// TIA Portal V21 export
FUNCTION_BLOCK "FB311"   // FB311, LAD
TITLE = FB311
{ S7_Optimized_Access := 'TRUE' }
AUTHOR : PRECISE
FAMILY : PRECISE
// TEMPERATURE CONTROL
// stored: AutoNumber false, MemoryReserve 100, SetENOAutomatically false
   VAR_INPUT
      Enable : Bool;
      Disable : Bool;
      Fault : Bool;
      SecPulse : Bool;
      AlwaysTrue : Bool;
      StartConfirmationPopupSel : Bool;   // StartConfirmationPopupSel: 0-NO/1-YES
      EndConfirmationPopupSel : Bool;   // EndConfirmationPopupSel: 0-NO/1-YES
      TimebaseSel : Bool;   // Timebase Selection: 0-sec/1-min
      TemperatureMaintainSel : Bool;   // Temperature Maintain Selection: 0-NO/1-YES
      BypassSel : Bool;   // Bypass Selection: 0-NO/1-YES
      JacketAirPurgingSel : Bool;   // Applicable for if Air Inlet Valve is present in jacket. 0-NO/1-YES
      TemperatureControlSel : Int;   // Temperature Control Sel : 0-Heat/1-Cool
      SensorSel : Int;   // Sensor Slection: 0-Vessel/1-Jacket
      BatchSizeSel : Int;   // Batch Size Sel:0-Small/1-Big
      HeatingUtilitySel : Int;   // Heating Utility Selection: 0-Steam/1-Hot Water
      CoolingUtilitySelection : Int;   // 0-cooling/1-chilling/2-brine/3-cooling+chilling/4-chilling+brine/5-cooling+chilling+Brine
      SetTemperature : Real := 60.0;
      TimeMin : Int := 1;   // For Temperature Maintain Selection: 1-YES & Bypass Selection: 1-YES
      TimeSec : Int := 30;   // For Temperature Maintain Selection: 1-YES & Bypass Selection: 0-NO
      ActualTemperatureVessel : Real;   // For Sensor Slection: 0-Vessel
      ActualTemperatureJacket : Real;   // For Sensor Slection: 1-Jacket
      JVDelay : Int := 5;
      JDDelay : Int := 5;
      TemperatureTol : Real := 0.3;
      CoolingThreshold : Real := 25.0;   // Temperature to change utility from cooling water to chilled water
      ChillingThreshold : Real := 15.0;   // Temperature to change utility from chilled water to brine water
      HeatHighTemperatureTol : Real := 3.0;
      CoolLowTemperatureTol : Real := 3.0;
      JacketAirPurgingTimeSec : Int := 10;
   END_VAR
   VAR_OUTPUT
      JacketAirValve : Bool;
      BypassValve : Bool;
      JacketVentValve1 : Bool;
      JacketDrainValve1 : Bool;
      CoolingWaterInletValve1 : Bool;
      CoolingWaterOutletValve1 : Bool;
      ChilledWaterInletValve1 : Bool;
      ChilledWaterOutletValve1 : Bool;
      BrineWaterInletValve1 : Bool;
      BrineWaterOutletValve1 : Bool;
      HotWaterInletValve1 : Bool;
      HotWaterOutletValve1 : Bool;
      SteamInlet1 : Bool;
      Condensateoutlet1 : Bool;
      JacketVentValve2 : Bool;
      JacketDrainValve2 : Bool;
      CoolingWaterInletValve2 : Bool;
      CoolingWaterOutletValve2 : Bool;
      ChilledWaterInletValve2 : Bool;
      ChilledWaterOutletValve2 : Bool;
      BrineWaterInletValve2 : Bool;
      BrineWaterOutletValve2 : Bool;
      HotWaterInletValve2 : Bool;
      HotWaterOutletValve2 : Bool;
      SteamInlet2 : Bool;
      Condensateoutlet2 : Bool;
      AlarmHeatHighTemperature : Bool;
      AlarmCoolLowTemperature : Bool;
      StartConfirmationPopup : Bool;   // For Start Confirmation Popup Selection: Yes
      EndConfirmationPopup : Bool;   // For End Confirmation Popup Selection: Yes
      JacketAirPurgingPopup : Bool;
      TimeMinPV : DInt;
      TimeSecPV : DInt;
      JacketAirPurgingTimeSecPV : Int;
      PrintTrigger : Bool;
      PrintWord : Int;
      PrintStatus : String[50];
   END_VAR
   VAR_IN_OUT
      Start : Bool;
      Stop : Bool;
      Reset : Bool;
      StartConfirmationAck : Bool;   // For Start Confirmation Popup Selection: Yes
      EndConfirmationAck : Bool;   // For End Confirmation Popup Selection: Yes
      JacketAirPurgingAck : Bool;
      AlarmAck : Bool;
      SpareBtn1 : Bool;
      Running : Bool;
      Selected : Bool;
      Paused : Bool;
      StartConfirmationPopupTemp : Bool;   // For Start Confirmation Popup Selection: Yes
      EndConfirmationPopupTemp : Bool;   // For End Confirmation Popup Selection: Yes
      Started : Bool;
      Over : Bool;
      StartJVDelay : Bool;
      StartJDDelay : Bool;
      StartUtility : Bool;
      StartChilling : Bool;
      StartBrine : Bool;
      StartJacketAirPurging : Bool;
      HeatTempReached : Bool;
      CoolTempReached : Bool;
      TemperatureTolNeg : Real;
      TemperatureTolPos : Real;
      HeatHighTemperatureTolCal : Real := 3.0;
      CoolLowTemperatureTolCal : Real := 3.0;
      JacketPressureSelection : Bool;   // 0-no,1-yes
      JacketPressureReached : Bool;
      JacketUtilityPressureValve : Bool;
      JAcketAlarms : Bool;
      Temp : Bool;
      JacketTime : Int;
      JacketSafetyPressure : Real;
      JAcketActPressure : Real;
   END_VAR
   VAR
      PrintTriggerTemp : Bool;
      RE1 : Bool;
      RE2 : Bool;
      RE3 : Bool;
      RE4 : Bool;
      RE5 : Bool;
      RE6 : Bool;
      RE7 : Bool;
      RE8 : Bool;
      RE9 : Bool;
      RE10 : Bool;
      RE11 : Bool;
      "Timer" : "FB101";
      PrintTriggerResetTimer { S7_SetPoint := 'True'} : TON_TIME;
      BtnResetTimer { S7_SetPoint := 'True'} : TON_TIME;
      JVDelayTime { S7_SetPoint := 'True'} : "FB103";
      JDDelayTime { S7_SetPoint := 'True'} : "FB103";
      JAPTime { S7_SetPoint := 'True'} : "FB103";
      ActualTemperature : Real;
      JacketpressureTimer { S7_SetPoint := 'True'} : "FB103";
      FB101_Instance { S7_SetPoint := 'True'} : "FB101";
   END_VAR
   VAR_TEMP
      STATUS1 : String[40];
      STATUS2 : String[40];
      STATUS3 : String[40];
      STATUS4 : String[40];
      STATUS5 : String[40];
      STATUS6 : String[40];
   END_VAR
   VAR_TEMP   // added for the SCL form of the ladder/FBD networks
      _w1 : Bool;
      _w2 : Bool;
      _w3 : Bool;
      _w4 : Bool;
      _w5 : Bool;
      _w6 : Bool;
      _w7 : Bool;
      _w8 : Bool;
   END_VAR
BEGIN

REGION Network 1: Running
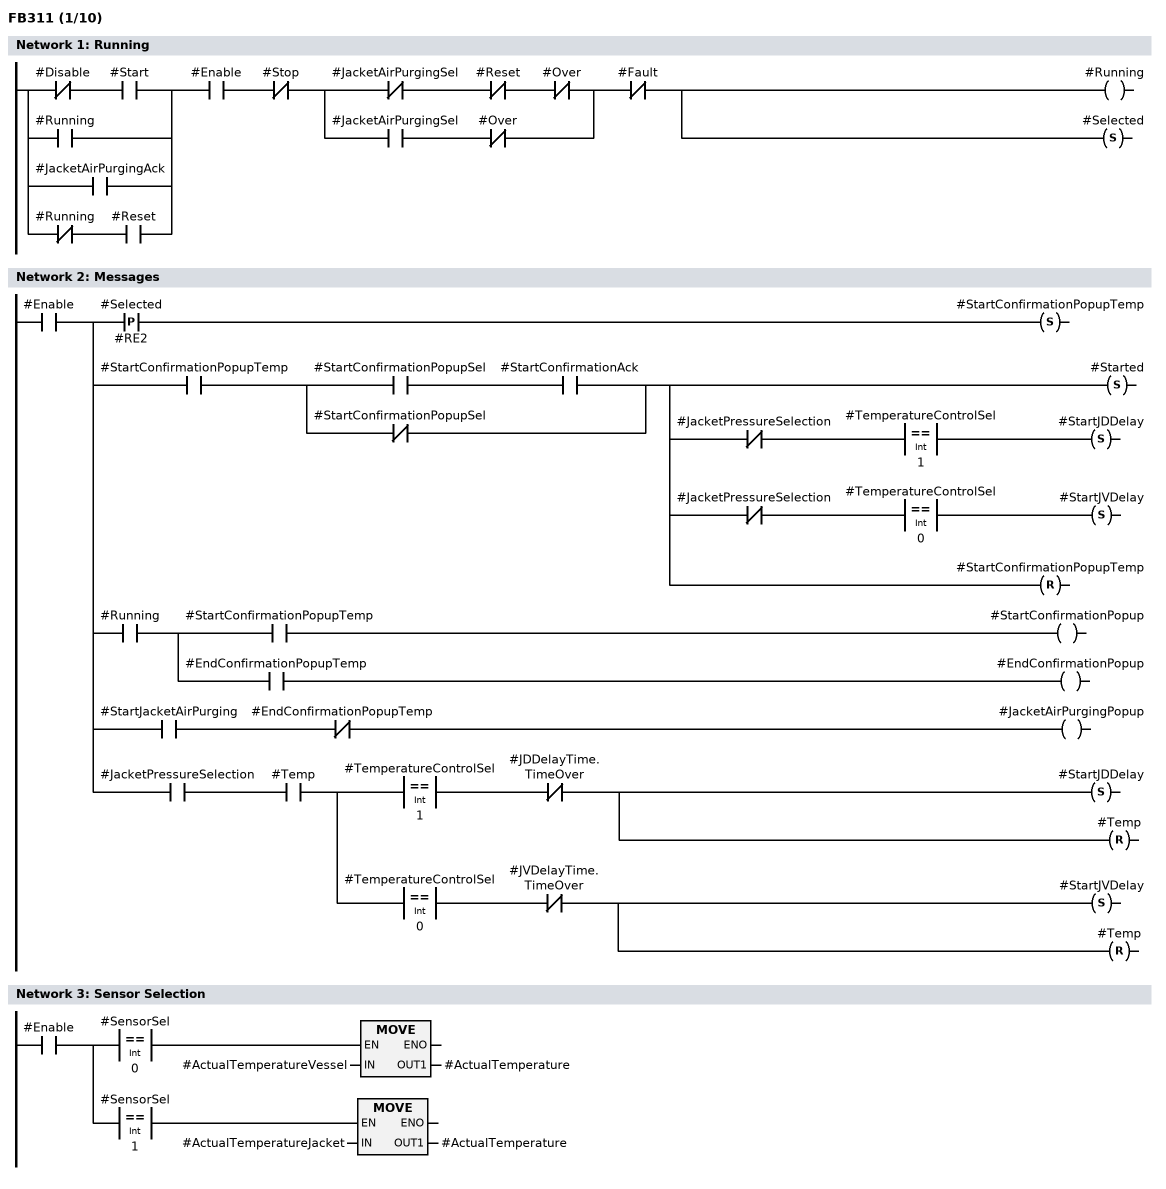
   RUNG wire#powerrail
      I_Contact( #Disable )
      Contact( #Start )
      wire#w1
      Contact( #Enable )
      I_Contact( #Stop )
      wire#w2
      I_Contact( #JacketAirPurgingSel )
      I_Contact( #Reset )
      I_Contact( #Over )
      wire#w3
      I_Contact( #Fault )
      wire#w4
      Coil( #Running )
   END_RUNG
   RUNG wire#powerrail
      Contact( #Running )
   END_RUNG wire#w1
   RUNG wire#powerrail
      Contact( #JacketAirPurgingAck )
   END_RUNG wire#w1
   RUNG wire#powerrail
      I_Contact( #Running )
      Contact( #Reset )
   END_RUNG wire#w1
   RUNG wire#w2
      Contact( #JacketAirPurgingSel )
      I_Contact( #Over )
   END_RUNG wire#w3
   RUNG wire#w4
      S_Coil( #Selected )
   END_RUNG
   // the same network as SCL:
   #Running := ((NOT #Disable AND #Start) OR #Running OR #JacketAirPurgingAck OR (NOT #Running AND #Reset)) AND #Enable AND NOT #Stop AND ((NOT #JacketAirPurgingSel AND NOT #Reset AND NOT #Over) OR (#JacketAirPurgingSel AND NOT #Over)) AND NOT #Fault;
   IF #Running THEN #Selected := TRUE; END_IF;
END_REGION

REGION Network 2: Messages
   RUNG wire#powerrail
      Contact( #Enable )
      wire#w1
      P_Contact(operand := #Selected, bit := #RE2)
      S_Coil( #StartConfirmationPopupTemp )
   END_RUNG
   RUNG wire#w1
      Contact( #StartConfirmationPopupTemp )
      wire#w2
      Contact( #StartConfirmationPopupSel )
      Contact( #StartConfirmationAck )
      wire#w3
      S_Coil( #Started )
   END_RUNG
   RUNG wire#w2
      I_Contact( #StartConfirmationPopupSel )
   END_RUNG wire#w3
   RUNG wire#w3
      I_Contact( #JacketPressureSelection )
      { S7_Templates := "SrcType := Int" } EQ_Contact(in1 := #TemperatureControlSel, in2 := 1)
      S_Coil( #StartJDDelay )
   END_RUNG
   RUNG wire#w3
      I_Contact( #JacketPressureSelection )
      { S7_Templates := "SrcType := Int" } EQ_Contact(in1 := #TemperatureControlSel, in2 := 0)
      S_Coil( #StartJVDelay )
   END_RUNG
   RUNG wire#w3
      R_Coil( #StartConfirmationPopupTemp )
   END_RUNG
   RUNG wire#w1
      Contact( #Running )
      wire#w4
      Contact( #StartConfirmationPopupTemp )
      Coil( #StartConfirmationPopup )
   END_RUNG
   RUNG wire#w4
      Contact( #EndConfirmationPopupTemp )
      Coil( #EndConfirmationPopup )
   END_RUNG
   RUNG wire#w1
      Contact( #StartJacketAirPurging )
      I_Contact( #EndConfirmationPopupTemp )
      Coil( #JacketAirPurgingPopup )
   END_RUNG
   RUNG wire#w1
      Contact( #JacketPressureSelection )
      Contact( #Temp )
      wire#w5
      { S7_Templates := "SrcType := Int" } EQ_Contact(in1 := #TemperatureControlSel, in2 := 1)
      I_Contact( #JDDelayTime.TimeOver )
      wire#w6
      S_Coil( #StartJDDelay )
   END_RUNG
   RUNG wire#w6
      R_Coil( #Temp )
   END_RUNG
   RUNG wire#w5
      { S7_Templates := "SrcType := Int" } EQ_Contact(in1 := #TemperatureControlSel, in2 := 0)
      I_Contact( #JVDelayTime.TimeOver )
      wire#w7
      S_Coil( #StartJVDelay )
   END_RUNG
   RUNG wire#w7
      R_Coil( #Temp )
   END_RUNG
   // the same network as SCL:
   #_w1 := #Enable AND #Selected AND NOT #RE2;   // rising edge of #Selected
   #RE2 := #Selected;
   IF #_w1 THEN #StartConfirmationPopupTemp := TRUE; END_IF;
   #_w2 := #Enable AND #StartConfirmationPopupTemp AND ((#StartConfirmationPopupSel AND #StartConfirmationAck) OR NOT #StartConfirmationPopupSel);
   IF #_w2 THEN #Started := TRUE; END_IF;
   IF #_w2 AND NOT #JacketPressureSelection AND (#TemperatureControlSel = 1) THEN
       #StartJDDelay := TRUE;
   END_IF;
   IF #_w2 AND NOT #JacketPressureSelection AND (#TemperatureControlSel = 0) THEN
       #StartJVDelay := TRUE;
   END_IF;
   IF #_w2 THEN #StartConfirmationPopupTemp := FALSE; END_IF;
   #_w3 := #Enable AND #Running;
   #StartConfirmationPopup := #_w3 AND #StartConfirmationPopupTemp;
   #EndConfirmationPopup := #_w3 AND #EndConfirmationPopupTemp;
   #JacketAirPurgingPopup := #Enable AND #StartJacketAirPurging AND NOT #EndConfirmationPopupTemp;
   #_w4 := #Enable AND #JacketPressureSelection AND #Temp;
   IF #_w4 AND (#TemperatureControlSel = 1) AND NOT #JDDelayTime.TimeOver THEN
       #StartJDDelay := TRUE;
       #Temp := FALSE;
   END_IF;
   IF #_w4 AND (#TemperatureControlSel = 0) AND NOT #JVDelayTime.TimeOver THEN
       #StartJVDelay := TRUE;
       #Temp := FALSE;
   END_IF;
END_REGION

REGION Network 3: Sensor Selection
   RUNG wire#powerrail
      Contact( #Enable )
      wire#w1
      { S7_Templates := "SrcType := Int" } EQ_Contact(in1 := #SensorSel, in2 := 0)
      Move(in := #ActualTemperatureVessel, out1 => #ActualTemperature)
   END_RUNG
   RUNG wire#w1
      { S7_Templates := "SrcType := Int" } EQ_Contact(in1 := #SensorSel, in2 := 1)
      Move(in := #ActualTemperatureJacket, out1 => #ActualTemperature)
   END_RUNG
   // the same network as SCL:
   IF #Enable AND (#SensorSel = 0) THEN #ActualTemperature := #ActualTemperatureVessel; END_IF;
   IF #Enable AND (#SensorSel = 1) THEN #ActualTemperature := #ActualTemperatureJacket; END_IF;
END_REGION

REGION Network 4: Tolerance
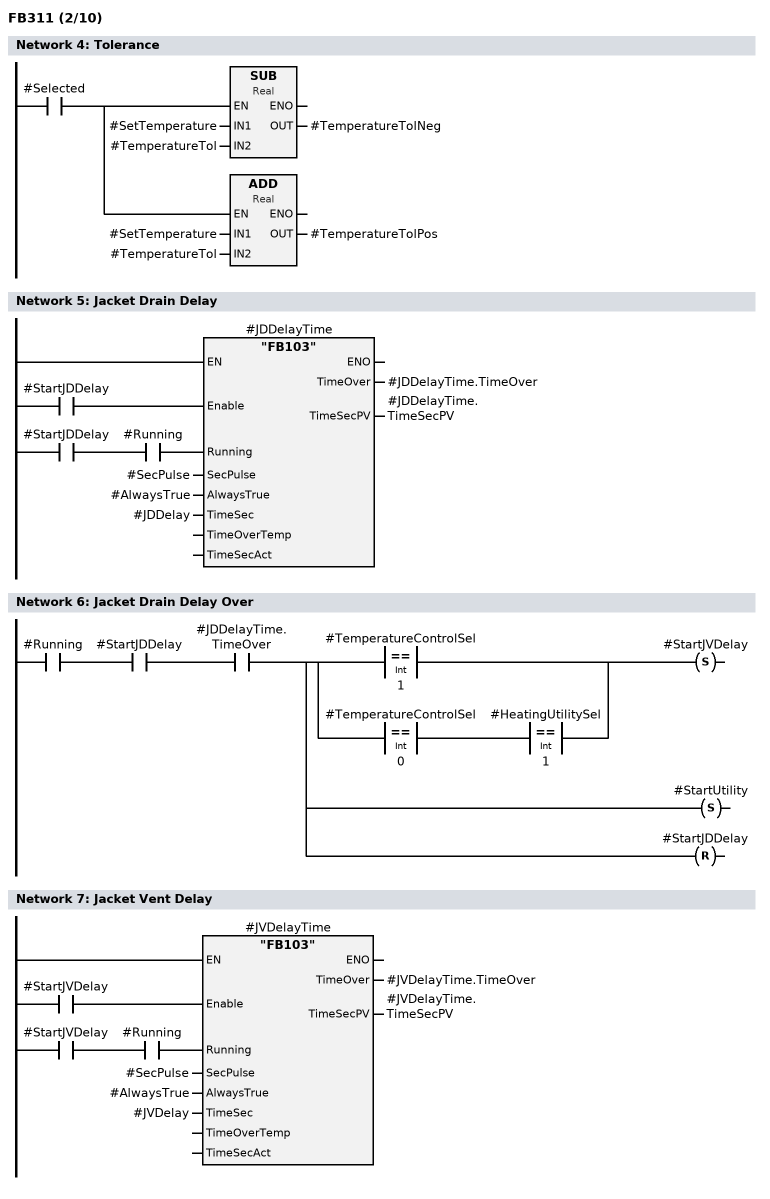
   RUNG wire#powerrail
      Contact( #Selected )
      wire#w1
      { S7_Templates := "SrcType := Real"; S7_GenerateENO := "TRUE" } Sub(in1 := #SetTemperature, in2 := #TemperatureTol, out => #TemperatureTolNeg)
   END_RUNG
   RUNG wire#w1
      { S7_Templates := "SrcType := Real"; S7_GenerateENO := "TRUE" } Add(in1 := #SetTemperature, in2 := #TemperatureTol, out => #TemperatureTolPos)
   END_RUNG
   // the same network as SCL:
   IF #Selected THEN
       #TemperatureTolNeg := #SetTemperature - #TemperatureTol;
       #TemperatureTolPos := #SetTemperature + #TemperatureTol;
   END_IF;
END_REGION

REGION Network 5: Jacket Drain Delay
   RUNG wire#powerrail
      #JDDelayTime(Enable := wire#w1, Running := wire#w2, SecPulse := #SecPulse, AlwaysTrue := #AlwaysTrue, TimeSec := #JDDelay, TimeOverTemp :=, TimeSecAct :=, TimeOver => #JDDelayTime.TimeOver, TimeSecPV => #JDDelayTime.TimeSecPV)
   END_RUNG
   RUNG wire#powerrail
      Contact( #StartJDDelay )
   END_RUNG wire#w1
   RUNG wire#powerrail
      Contact( #StartJDDelay )
      Contact( #Running )
   END_RUNG wire#w2
   // the same network as SCL:
   #JDDelayTime(Enable := #StartJDDelay,   // "FB103"
                Running := #StartJDDelay AND #Running,
                SecPulse := #SecPulse,
                AlwaysTrue := #AlwaysTrue,
                TimeSec := #JDDelay,
                TimeOver => #JDDelayTime.TimeOver,
                TimeSecPV => #JDDelayTime.TimeSecPV);
END_REGION

REGION Network 6: Jacket Drain Delay Over
   RUNG wire#powerrail
      Contact( #Running )
      Contact( #StartJDDelay )
      Contact( #JDDelayTime.TimeOver )
      wire#w1
      { S7_Templates := "SrcType := Int" } EQ_Contact(in1 := #TemperatureControlSel, in2 := 1)
      wire#w2
      S_Coil( #StartJVDelay )
   END_RUNG
   RUNG wire#w1
      { S7_Templates := "SrcType := Int" } EQ_Contact(in1 := #TemperatureControlSel, in2 := 0)
      { S7_Templates := "SrcType := Int" } EQ_Contact(in1 := #HeatingUtilitySel, in2 := 1)
   END_RUNG wire#w2
   RUNG wire#w1
      S_Coil( #StartUtility )
   END_RUNG
   RUNG wire#w1
      R_Coil( #StartJDDelay )
   END_RUNG
   // the same network as SCL:
   #_w1 := #Running AND #StartJDDelay AND #JDDelayTime.TimeOver;
   IF #_w1 AND ((#TemperatureControlSel = 1) OR ((#TemperatureControlSel = 0) AND (#HeatingUtilitySel = 1))) THEN
       #StartJVDelay := TRUE;
   END_IF;
   IF #_w1 THEN
       #StartUtility := TRUE;
       #StartJDDelay := FALSE;
   END_IF;
END_REGION

REGION Network 7: Jacket Vent Delay
   RUNG wire#powerrail
      #JVDelayTime(Enable := wire#w1, Running := wire#w2, SecPulse := #SecPulse, AlwaysTrue := #AlwaysTrue, TimeSec := #JVDelay, TimeOverTemp :=, TimeSecAct :=, TimeOver => #JVDelayTime.TimeOver, TimeSecPV => #JVDelayTime.TimeSecPV)
   END_RUNG
   RUNG wire#powerrail
      Contact( #StartJVDelay )
   END_RUNG wire#w1
   RUNG wire#powerrail
      Contact( #StartJVDelay )
      Contact( #Running )
   END_RUNG wire#w2
   // the same network as SCL:
   #JVDelayTime(Enable := #StartJVDelay,   // "FB103"
                Running := #StartJVDelay AND #Running,
                SecPulse := #SecPulse,
                AlwaysTrue := #AlwaysTrue,
                TimeSec := #JVDelay,
                TimeOver => #JVDelayTime.TimeOver,
                TimeSecPV => #JVDelayTime.TimeSecPV);
END_REGION

REGION Network 8: Jacket Vent Delay Over
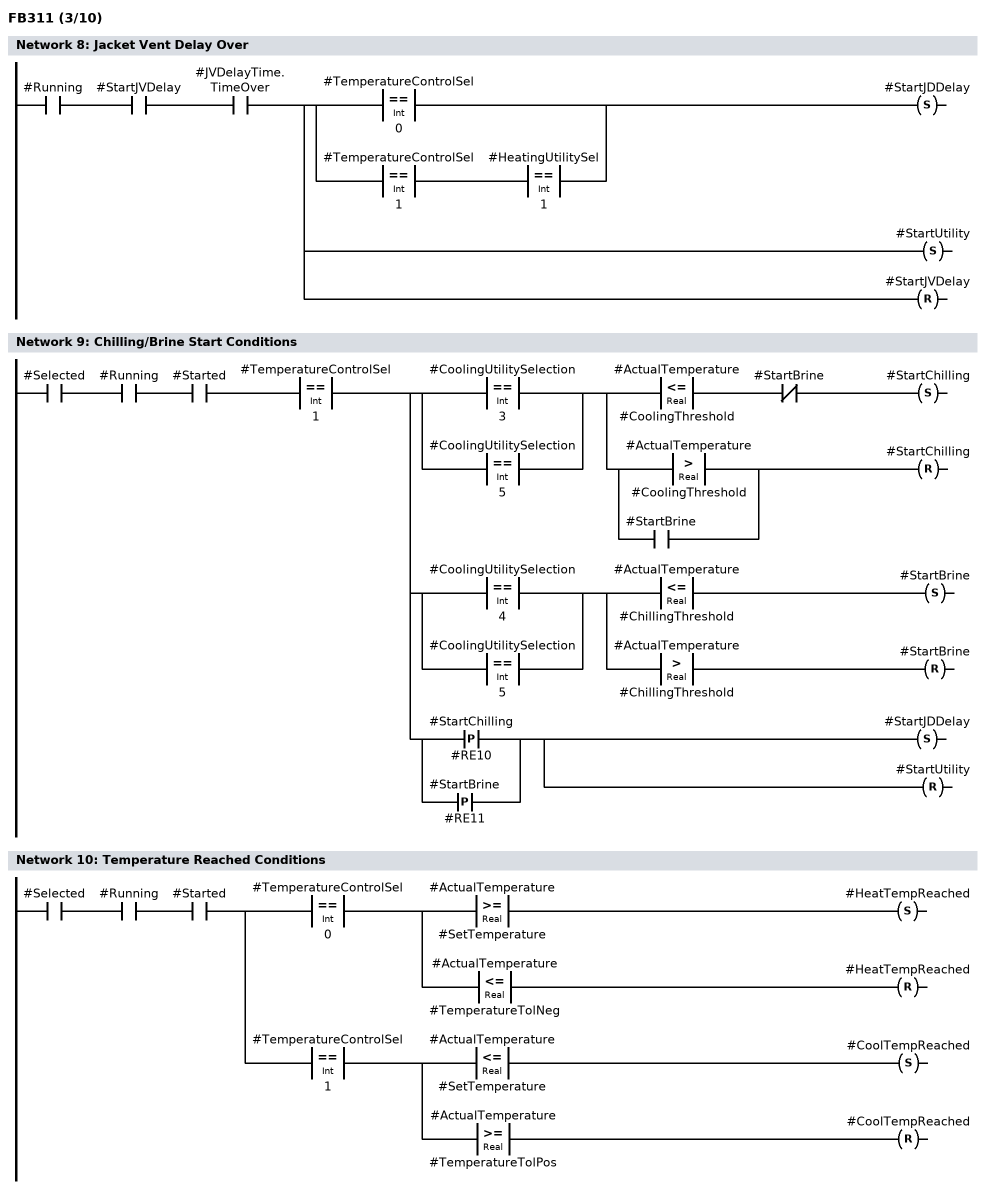
   RUNG wire#powerrail
      Contact( #Running )
      Contact( #StartJVDelay )
      Contact( #JVDelayTime.TimeOver )
      wire#w1
      { S7_Templates := "SrcType := Int" } EQ_Contact(in1 := #TemperatureControlSel, in2 := 0)
      wire#w2
      S_Coil( #StartJDDelay )
   END_RUNG
   RUNG wire#w1
      { S7_Templates := "SrcType := Int" } EQ_Contact(in1 := #TemperatureControlSel, in2 := 1)
      { S7_Templates := "SrcType := Int" } EQ_Contact(in1 := #HeatingUtilitySel, in2 := 1)
   END_RUNG wire#w2
   RUNG wire#w1
      S_Coil( #StartUtility )
   END_RUNG
   RUNG wire#w1
      R_Coil( #StartJVDelay )
   END_RUNG
   // the same network as SCL:
   #_w1 := #Running AND #StartJVDelay AND #JVDelayTime.TimeOver;
   IF #_w1 AND ((#TemperatureControlSel = 0) OR ((#TemperatureControlSel = 1) AND (#HeatingUtilitySel = 1))) THEN
       #StartJDDelay := TRUE;
   END_IF;
   IF #_w1 THEN
       #StartUtility := TRUE;
       #StartJVDelay := FALSE;
   END_IF;
END_REGION

REGION Network 9: Chilling/Brine Start Conditions
   RUNG wire#powerrail
      Contact( #Selected )
      Contact( #Running )
      Contact( #Started )
      { S7_Templates := "SrcType := Int" } EQ_Contact(in1 := #TemperatureControlSel, in2 := 1)
      wire#w1
      { S7_Templates := "SrcType := Int" } EQ_Contact(in1 := #CoolingUtilitySelection, in2 := 3)
      wire#w2
      { S7_Templates := "SrcType := Real" } LE_Contact(in1 := #ActualTemperature, in2 := #CoolingThreshold)
      I_Contact( #StartBrine )
      S_Coil( #StartChilling )
   END_RUNG
   RUNG wire#w1
      { S7_Templates := "SrcType := Int" } EQ_Contact(in1 := #CoolingUtilitySelection, in2 := 5)
   END_RUNG wire#w2
   RUNG wire#w2
      { S7_Templates := "SrcType := Real" } GT_Contact(in1 := #ActualTemperature, in2 := #CoolingThreshold)
      wire#w3
      R_Coil( #StartChilling )
   END_RUNG
   RUNG wire#w2
      Contact( #StartBrine )
   END_RUNG wire#w3
   RUNG wire#w1
      { S7_Templates := "SrcType := Int" } EQ_Contact(in1 := #CoolingUtilitySelection, in2 := 4)
      wire#w4
      { S7_Templates := "SrcType := Real" } LE_Contact(in1 := #ActualTemperature, in2 := #ChillingThreshold)
      S_Coil( #StartBrine )
   END_RUNG
   RUNG wire#w1
      { S7_Templates := "SrcType := Int" } EQ_Contact(in1 := #CoolingUtilitySelection, in2 := 5)
   END_RUNG wire#w4
   RUNG wire#w4
      { S7_Templates := "SrcType := Real" } GT_Contact(in1 := #ActualTemperature, in2 := #ChillingThreshold)
      R_Coil( #StartBrine )
   END_RUNG
   RUNG wire#w1
      P_Contact(operand := #StartChilling, bit := #RE10)
      wire#w5
      S_Coil( #StartJDDelay )
   END_RUNG
   RUNG wire#w1
      P_Contact(operand := #StartBrine, bit := #RE11)
   END_RUNG wire#w5
   RUNG wire#w5
      R_Coil( #StartUtility )
   END_RUNG
   // the same network as SCL:
   #_w1 := #Selected AND #Running AND #Started AND (#TemperatureControlSel = 1);
   #_w2 := #_w1 AND ((#CoolingUtilitySelection = 3) OR (#CoolingUtilitySelection = 5));
   IF #_w2 AND (#ActualTemperature <= #CoolingThreshold) AND NOT #StartBrine THEN
       #StartChilling := TRUE;
   END_IF;
   IF #_w2 AND ((#ActualTemperature > #CoolingThreshold) OR #StartBrine) THEN
       #StartChilling := FALSE;
   END_IF;
   #_w3 := #_w1 AND ((#CoolingUtilitySelection = 4) OR (#CoolingUtilitySelection = 5));
   IF #_w3 AND (#ActualTemperature <= #ChillingThreshold) THEN #StartBrine := TRUE; END_IF;
   IF #_w3 AND (#ActualTemperature > #ChillingThreshold) THEN #StartBrine := FALSE; END_IF;
   #_w4 := #_w1 AND #StartChilling AND NOT #RE10;   // rising edge of #StartChilling
   #RE10 := #StartChilling;
   #_w5 := #_w1 AND #StartBrine AND NOT #RE11;   // rising edge of #StartBrine
   #RE11 := #StartBrine;
   IF #_w4 OR #_w5 THEN
       #StartJDDelay := TRUE;
       #StartUtility := FALSE;
   END_IF;
END_REGION

REGION Network 10: Temperature Reached Conditions
   RUNG wire#powerrail
      Contact( #Selected )
      Contact( #Running )
      Contact( #Started )
      wire#w1
      { S7_Templates := "SrcType := Int" } EQ_Contact(in1 := #TemperatureControlSel, in2 := 0)
      wire#w2
      { S7_Templates := "SrcType := Real" } GE_Contact(in1 := #ActualTemperature, in2 := #SetTemperature)
      S_Coil( #HeatTempReached )
   END_RUNG
   RUNG wire#w2
      { S7_Templates := "SrcType := Real" } LE_Contact(in1 := #ActualTemperature, in2 := #TemperatureTolNeg)
      R_Coil( #HeatTempReached )
   END_RUNG
   RUNG wire#w1
      { S7_Templates := "SrcType := Int" } EQ_Contact(in1 := #TemperatureControlSel, in2 := 1)
      wire#w3
      { S7_Templates := "SrcType := Real" } LE_Contact(in1 := #ActualTemperature, in2 := #SetTemperature)
      S_Coil( #CoolTempReached )
   END_RUNG
   RUNG wire#w3
      { S7_Templates := "SrcType := Real" } GE_Contact(in1 := #ActualTemperature, in2 := #TemperatureTolPos)
      R_Coil( #CoolTempReached )
   END_RUNG
   // the same network as SCL:
   #_w1 := #Selected AND #Running AND #Started;
   #_w2 := #_w1 AND (#TemperatureControlSel = 0);
   IF #_w2 AND (#ActualTemperature >= #SetTemperature) THEN #HeatTempReached := TRUE; END_IF;
   IF #_w2 AND (#ActualTemperature <= #TemperatureTolNeg) THEN #HeatTempReached := FALSE; END_IF;
   #_w3 := #_w1 AND (#TemperatureControlSel = 1);
   IF #_w3 AND (#ActualTemperature <= #SetTemperature) THEN #CoolTempReached := TRUE; END_IF;
   IF #_w3 AND (#ActualTemperature >= #TemperatureTolPos) THEN #CoolTempReached := FALSE; END_IF;
END_REGION

REGION Network 11: Timer
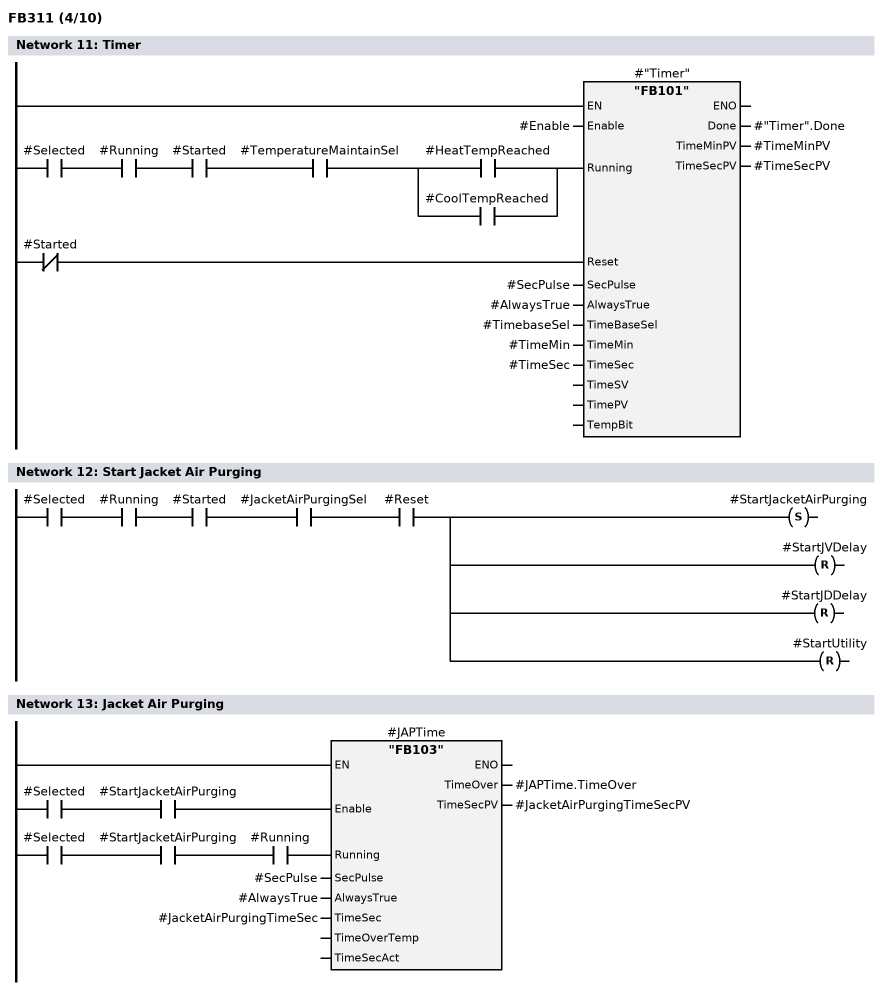
   RUNG wire#powerrail
      #"Timer"(Running := wire#w2, Reset := wire#w3, Enable := #Enable, SecPulse := #SecPulse, AlwaysTrue := #AlwaysTrue, TimeBaseSel := #TimebaseSel, TimeMin := #TimeMin, TimeSec := #TimeSec, TimeSV :=, TimePV :=, TempBit :=, Done => #"Timer".Done, TimeMinPV => #TimeMinPV, TimeSecPV => #TimeSecPV)
   END_RUNG
   RUNG wire#powerrail
      Contact( #Selected )
      Contact( #Running )
      Contact( #Started )
      Contact( #TemperatureMaintainSel )
      wire#w1
      Contact( #HeatTempReached )
   END_RUNG wire#w2
   RUNG wire#w1
      Contact( #CoolTempReached )
   END_RUNG wire#w2
   RUNG wire#powerrail
      I_Contact( #Started )
   END_RUNG wire#w3
   // the same network as SCL:
   #"Timer"(Enable := #Enable,   // "FB101"
            Running := #Selected AND #Running AND #Started AND #TemperatureMaintainSel AND (#HeatTempReached OR #CoolTempReached),
            Reset := NOT #Started,
            SecPulse := #SecPulse,
            AlwaysTrue := #AlwaysTrue,
            TimeBaseSel := #TimebaseSel,
            TimeMin := #TimeMin,
            TimeSec := #TimeSec,
            Done => #"Timer".Done,
            TimeMinPV => #TimeMinPV,
            TimeSecPV => #TimeSecPV);
END_REGION

REGION Network 12: Start Jacket Air Purging
   RUNG wire#powerrail
      Contact( #Selected )
      Contact( #Running )
      Contact( #Started )
      Contact( #JacketAirPurgingSel )
      Contact( #Reset )
      wire#w1
      S_Coil( #StartJacketAirPurging )
   END_RUNG
   RUNG wire#w1
      R_Coil( #StartJVDelay )
   END_RUNG
   RUNG wire#w1
      R_Coil( #StartJDDelay )
   END_RUNG
   RUNG wire#w1
      R_Coil( #StartUtility )
   END_RUNG
   // the same network as SCL:
   IF #Selected AND #Running AND #Started AND #JacketAirPurgingSel AND #Reset THEN
       #StartJacketAirPurging := TRUE;
       #StartJVDelay := FALSE;
       #StartJDDelay := FALSE;
       #StartUtility := FALSE;
   END_IF;
END_REGION

REGION Network 13: Jacket Air Purging
   RUNG wire#powerrail
      #JAPTime(Enable := wire#w1, Running := wire#w2, SecPulse := #SecPulse, AlwaysTrue := #AlwaysTrue, TimeSec := #JacketAirPurgingTimeSec, TimeOverTemp :=, TimeSecAct :=, TimeOver => #JAPTime.TimeOver, TimeSecPV => #JacketAirPurgingTimeSecPV)
   END_RUNG
   RUNG wire#powerrail
      Contact( #Selected )
      Contact( #StartJacketAirPurging )
   END_RUNG wire#w1
   RUNG wire#powerrail
      Contact( #Selected )
      Contact( #StartJacketAirPurging )
      Contact( #Running )
   END_RUNG wire#w2
   // the same network as SCL:
   #JAPTime(Enable := #Selected AND #StartJacketAirPurging,   // "FB103"
            Running := #Selected AND #StartJacketAirPurging AND #Running,
            SecPulse := #SecPulse,
            AlwaysTrue := #AlwaysTrue,
            TimeSec := #JacketAirPurgingTimeSec,
            TimeOver => #JAPTime.TimeOver,
            TimeSecPV => #JacketAirPurgingTimeSecPV);
END_REGION

REGION Network 14: Over
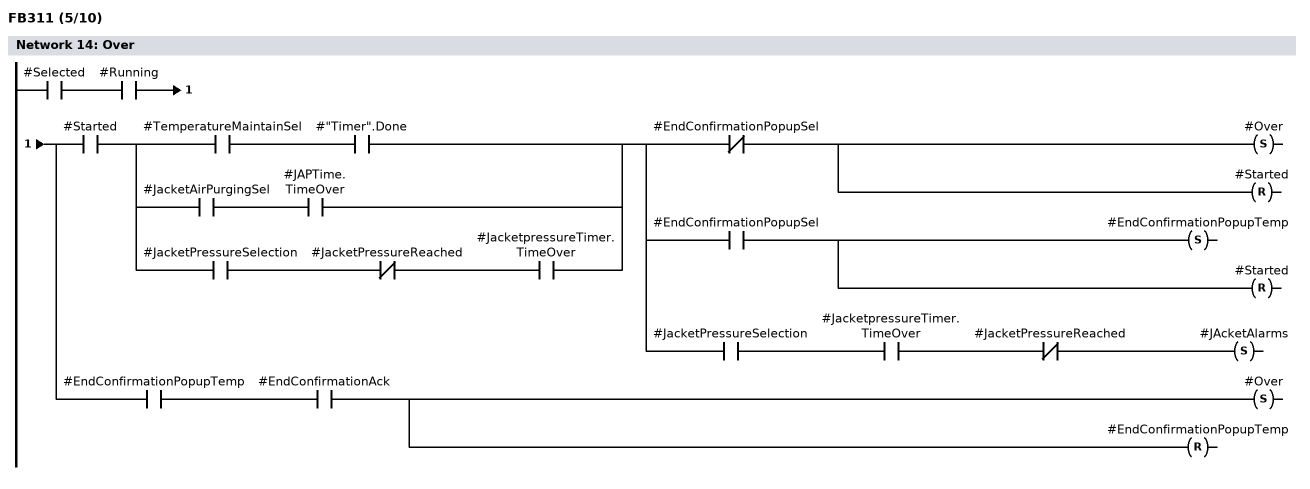
   RUNG wire#powerrail
      Contact( #Selected )
      Contact( #Running )
      wire#w1
      Contact( #Started )
      wire#w2
      Contact( #TemperatureMaintainSel )
      Contact( #"Timer".Done )
      wire#w3
      I_Contact( #EndConfirmationPopupSel )
      wire#w4
      S_Coil( #Over )
   END_RUNG
   RUNG wire#w2
      Contact( #JacketAirPurgingSel )
      Contact( #JAPTime.TimeOver )
   END_RUNG wire#w3
   RUNG wire#w2
      Contact( #JacketPressureSelection )
      I_Contact( #JacketPressureReached )
      Contact( #JacketpressureTimer.TimeOver )
   END_RUNG wire#w3
   RUNG wire#w4
      R_Coil( #Started )
   END_RUNG
   RUNG wire#w3
      Contact( #EndConfirmationPopupSel )
      wire#w5
      S_Coil( #EndConfirmationPopupTemp )
   END_RUNG
   RUNG wire#w5
      R_Coil( #Started )
   END_RUNG
   RUNG wire#w3
      Contact( #JacketPressureSelection )
      Contact( #JacketpressureTimer.TimeOver )
      I_Contact( #JacketPressureReached )
      S_Coil( #JAcketAlarms )
   END_RUNG
   RUNG wire#w1
      Contact( #EndConfirmationPopupTemp )
      Contact( #EndConfirmationAck )
      wire#w6
      S_Coil( #Over )
   END_RUNG
   RUNG wire#w6
      R_Coil( #EndConfirmationPopupTemp )
   END_RUNG
   // the same network as SCL:
   #_w1 := #Selected AND #Running;
   #_w2 := #_w1 AND #Started AND ((#TemperatureMaintainSel AND #"Timer".Done) OR (#JacketAirPurgingSel AND #JAPTime.TimeOver) OR (#JacketPressureSelection AND NOT #JacketPressureReached AND #JacketpressureTimer.TimeOver));
   IF #_w2 AND NOT #EndConfirmationPopupSel THEN
       #Over := TRUE;
       #Started := FALSE;
   END_IF;
   IF #_w2 AND #EndConfirmationPopupSel THEN
       #EndConfirmationPopupTemp := TRUE;
       #Started := FALSE;
   END_IF;
   IF #_w2 AND #JacketPressureSelection AND #JacketpressureTimer.TimeOver AND NOT #JacketPressureReached THEN
       #JAcketAlarms := TRUE;
   END_IF;
   IF #_w1 AND #EndConfirmationPopupTemp AND #EndConfirmationAck THEN
       #Over := TRUE;
       #EndConfirmationPopupTemp := FALSE;
   END_IF;
END_REGION

REGION Network 15: Outputs
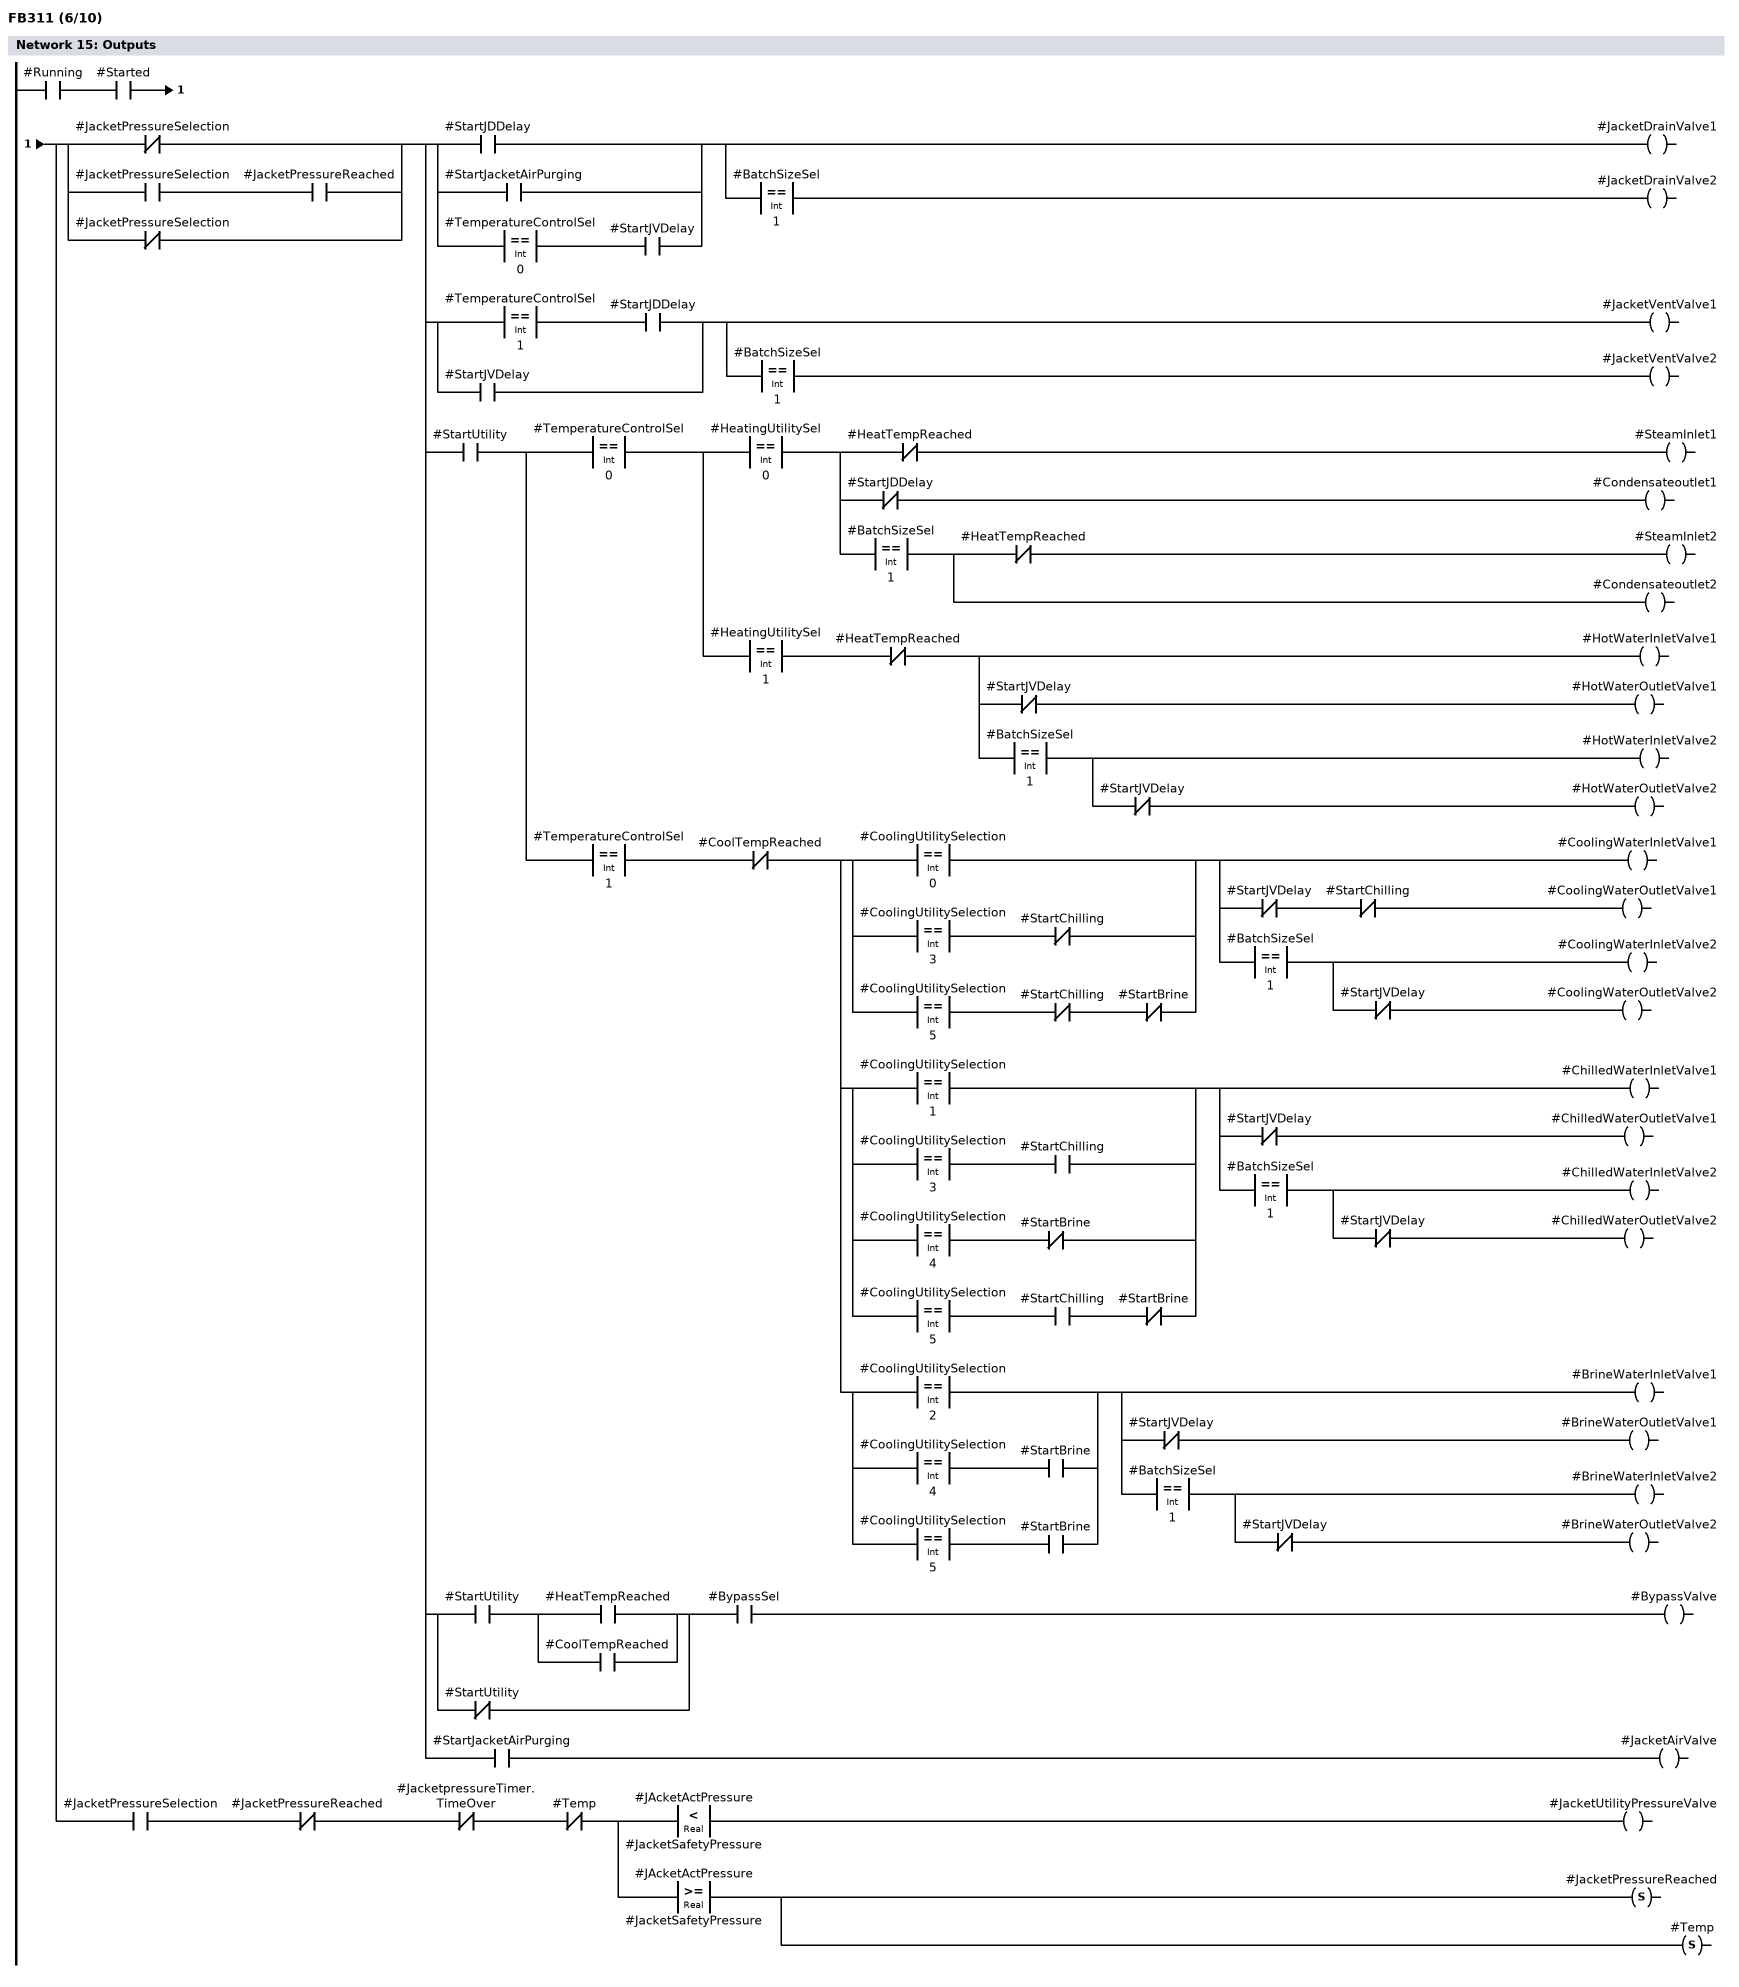
   RUNG wire#powerrail
      Contact( #Running )
      Contact( #Started )
      wire#w1
      I_Contact( #JacketPressureSelection )
      wire#w2
      Contact( #StartJDDelay )
      wire#w3
      Coil( #JacketDrainValve1 )
   END_RUNG
   RUNG wire#w1
      Contact( #JacketPressureSelection )
      Contact( #JacketPressureReached )
   END_RUNG wire#w2
   RUNG wire#w1
      I_Contact( #JacketPressureSelection )
   END_RUNG wire#w2
   RUNG wire#w2
      Contact( #StartJacketAirPurging )
   END_RUNG wire#w3
   RUNG wire#w2
      { S7_Templates := "SrcType := Int" } EQ_Contact(in1 := #TemperatureControlSel, in2 := 0)
      Contact( #StartJVDelay )
   END_RUNG wire#w3
   RUNG wire#w3
      { S7_Templates := "SrcType := Int" } EQ_Contact(in1 := #BatchSizeSel, in2 := 1)
      Coil( #JacketDrainValve2 )
   END_RUNG
   RUNG wire#w2
      { S7_Templates := "SrcType := Int" } EQ_Contact(in1 := #TemperatureControlSel, in2 := 1)
      Contact( #StartJDDelay )
      wire#w4
      Coil( #JacketVentValve1 )
   END_RUNG
   RUNG wire#w2
      Contact( #StartJVDelay )
   END_RUNG wire#w4
   RUNG wire#w4
      { S7_Templates := "SrcType := Int" } EQ_Contact(in1 := #BatchSizeSel, in2 := 1)
      Coil( #JacketVentValve2 )
   END_RUNG
   RUNG wire#w2
      Contact( #StartUtility )
      wire#w5
      { S7_Templates := "SrcType := Int" } EQ_Contact(in1 := #TemperatureControlSel, in2 := 0)
      wire#w6
      { S7_Templates := "SrcType := Int" } EQ_Contact(in1 := #HeatingUtilitySel, in2 := 0)
      wire#w7
      I_Contact( #HeatTempReached )
      Coil( #SteamInlet1 )
   END_RUNG
   RUNG wire#w7
      I_Contact( #StartJDDelay )
      Coil( #Condensateoutlet1 )
   END_RUNG
   RUNG wire#w7
      { S7_Templates := "SrcType := Int" } EQ_Contact(in1 := #BatchSizeSel, in2 := 1)
      wire#w8
      I_Contact( #HeatTempReached )
      Coil( #SteamInlet2 )
   END_RUNG
   RUNG wire#w8
      Coil( #Condensateoutlet2 )
   END_RUNG
   RUNG wire#w6
      { S7_Templates := "SrcType := Int" } EQ_Contact(in1 := #HeatingUtilitySel, in2 := 1)
      I_Contact( #HeatTempReached )
      wire#w9
      Coil( #HotWaterInletValve1 )
   END_RUNG
   RUNG wire#w9
      I_Contact( #StartJVDelay )
      Coil( #HotWaterOutletValve1 )
   END_RUNG
   RUNG wire#w9
      { S7_Templates := "SrcType := Int" } EQ_Contact(in1 := #BatchSizeSel, in2 := 1)
      wire#w10
      Coil( #HotWaterInletValve2 )
   END_RUNG
   RUNG wire#w10
      I_Contact( #StartJVDelay )
      Coil( #HotWaterOutletValve2 )
   END_RUNG
   RUNG wire#w5
      { S7_Templates := "SrcType := Int" } EQ_Contact(in1 := #TemperatureControlSel, in2 := 1)
      I_Contact( #CoolTempReached )
      wire#w11
      { S7_Templates := "SrcType := Int" } EQ_Contact(in1 := #CoolingUtilitySelection, in2 := 0)
      wire#w12
      Coil( #CoolingWaterInletValve1 )
   END_RUNG
   RUNG wire#w11
      { S7_Templates := "SrcType := Int" } EQ_Contact(in1 := #CoolingUtilitySelection, in2 := 3)
      I_Contact( #StartChilling )
   END_RUNG wire#w12
   RUNG wire#w11
      { S7_Templates := "SrcType := Int" } EQ_Contact(in1 := #CoolingUtilitySelection, in2 := 5)
      I_Contact( #StartChilling )
      I_Contact( #StartBrine )
   END_RUNG wire#w12
   RUNG wire#w12
      I_Contact( #StartJVDelay )
      I_Contact( #StartChilling )
      Coil( #CoolingWaterOutletValve1 )
   END_RUNG
   RUNG wire#w12
      { S7_Templates := "SrcType := Int" } EQ_Contact(in1 := #BatchSizeSel, in2 := 1)
      wire#w13
      Coil( #CoolingWaterInletValve2 )
   END_RUNG
   RUNG wire#w13
      I_Contact( #StartJVDelay )
      Coil( #CoolingWaterOutletValve2 )
   END_RUNG
   RUNG wire#w11
      { S7_Templates := "SrcType := Int" } EQ_Contact(in1 := #CoolingUtilitySelection, in2 := 1)
      wire#w14
      Coil( #ChilledWaterInletValve1 )
   END_RUNG
   RUNG wire#w11
      { S7_Templates := "SrcType := Int" } EQ_Contact(in1 := #CoolingUtilitySelection, in2 := 3)
      Contact( #StartChilling )
   END_RUNG wire#w14
   RUNG wire#w11
      { S7_Templates := "SrcType := Int" } EQ_Contact(in1 := #CoolingUtilitySelection, in2 := 4)
      I_Contact( #StartBrine )
   END_RUNG wire#w14
   RUNG wire#w11
      { S7_Templates := "SrcType := Int" } EQ_Contact(in1 := #CoolingUtilitySelection, in2 := 5)
      Contact( #StartChilling )
      I_Contact( #StartBrine )
   END_RUNG wire#w14
   RUNG wire#w14
      I_Contact( #StartJVDelay )
      Coil( #ChilledWaterOutletValve1 )
   END_RUNG
   RUNG wire#w14
      { S7_Templates := "SrcType := Int" } EQ_Contact(in1 := #BatchSizeSel, in2 := 1)
      wire#w15
      Coil( #ChilledWaterInletValve2 )
   END_RUNG
   RUNG wire#w15
      I_Contact( #StartJVDelay )
      Coil( #ChilledWaterOutletValve2 )
   END_RUNG
   RUNG wire#w11
      { S7_Templates := "SrcType := Int" } EQ_Contact(in1 := #CoolingUtilitySelection, in2 := 2)
      wire#w16
      Coil( #BrineWaterInletValve1 )
   END_RUNG
   RUNG wire#w11
      { S7_Templates := "SrcType := Int" } EQ_Contact(in1 := #CoolingUtilitySelection, in2 := 4)
      Contact( #StartBrine )
   END_RUNG wire#w16
   RUNG wire#w11
      { S7_Templates := "SrcType := Int" } EQ_Contact(in1 := #CoolingUtilitySelection, in2 := 5)
      Contact( #StartBrine )
   END_RUNG wire#w16
   RUNG wire#w16
      I_Contact( #StartJVDelay )
      Coil( #BrineWaterOutletValve1 )
   END_RUNG
   RUNG wire#w16
      { S7_Templates := "SrcType := Int" } EQ_Contact(in1 := #BatchSizeSel, in2 := 1)
      wire#w17
      Coil( #BrineWaterInletValve2 )
   END_RUNG
   RUNG wire#w17
      I_Contact( #StartJVDelay )
      Coil( #BrineWaterOutletValve2 )
   END_RUNG
   RUNG wire#w2
      Contact( #StartUtility )
      wire#w18
      Contact( #HeatTempReached )
      wire#w19
      Contact( #BypassSel )
      Coil( #BypassValve )
   END_RUNG
   RUNG wire#w18
      Contact( #CoolTempReached )
   END_RUNG wire#w19
   RUNG wire#w2
      I_Contact( #StartUtility )
   END_RUNG wire#w19
   RUNG wire#w2
      Contact( #StartJacketAirPurging )
      Coil( #JacketAirValve )
   END_RUNG
   RUNG wire#w1
      Contact( #JacketPressureSelection )
      I_Contact( #JacketPressureReached )
      I_Contact( #JacketpressureTimer.TimeOver )
      I_Contact( #Temp )
      wire#w20
      { S7_Templates := "SrcType := Real" } LT_Contact(in1 := #JAcketActPressure, in2 := #JacketSafetyPressure)
      Coil( #JacketUtilityPressureValve )
   END_RUNG
   RUNG wire#w20
      { S7_Templates := "SrcType := Real" } GE_Contact(in1 := #JAcketActPressure, in2 := #JacketSafetyPressure)
      wire#w21
      S_Coil( #JacketPressureReached )
   END_RUNG
   RUNG wire#w21
      S_Coil( #Temp )
   END_RUNG
   // the same network as SCL:
   #_w1 := #Running AND #Started;
   #_w2 := #_w1 AND (NOT #JacketPressureSelection OR (#JacketPressureSelection AND #JacketPressureReached) OR NOT #JacketPressureSelection);
   #JacketDrainValve1 := #_w2 AND (#StartJDDelay OR #StartJacketAirPurging OR ((#TemperatureControlSel = 0) AND #StartJVDelay));
   #JacketDrainValve2 := #JacketDrainValve1 AND (#BatchSizeSel = 1);
   #JacketVentValve1 := #_w2 AND (((#TemperatureControlSel = 1) AND #StartJDDelay) OR #StartJVDelay);
   #JacketVentValve2 := #JacketVentValve1 AND (#BatchSizeSel = 1);
   #_w3 := #_w2 AND #StartUtility;
   #_w4 := #_w3 AND (#TemperatureControlSel = 0);
   #_w5 := #_w4 AND (#HeatingUtilitySel = 0);
   #SteamInlet1 := #_w5 AND NOT #HeatTempReached;
   #Condensateoutlet1 := #_w5 AND NOT #StartJDDelay;
   #_w6 := #_w5 AND (#BatchSizeSel = 1);
   #SteamInlet2 := #_w6 AND NOT #HeatTempReached;
   #Condensateoutlet2 := #_w6;
   #HotWaterInletValve1 := #_w4 AND (#HeatingUtilitySel = 1) AND NOT #HeatTempReached;
   #HotWaterOutletValve1 := #HotWaterInletValve1 AND NOT #StartJVDelay;
   #HotWaterInletValve2 := #HotWaterInletValve1 AND (#BatchSizeSel = 1);
   #HotWaterOutletValve2 := #HotWaterInletValve2 AND NOT #StartJVDelay;
   #_w7 := #_w3 AND (#TemperatureControlSel = 1) AND NOT #CoolTempReached;
   #CoolingWaterInletValve1 := #_w7 AND ((#CoolingUtilitySelection = 0) OR ((#CoolingUtilitySelection = 3) AND NOT #StartChilling) OR ((#CoolingUtilitySelection = 5) AND NOT #StartChilling AND NOT #StartBrine));
   #CoolingWaterOutletValve1 := #CoolingWaterInletValve1 AND NOT #StartJVDelay AND NOT #StartChilling;
   #CoolingWaterInletValve2 := #CoolingWaterInletValve1 AND (#BatchSizeSel = 1);
   #CoolingWaterOutletValve2 := #CoolingWaterInletValve2 AND NOT #StartJVDelay;
   #ChilledWaterInletValve1 := #_w7 AND ((#CoolingUtilitySelection = 1) OR ((#CoolingUtilitySelection = 3) AND #StartChilling) OR ((#CoolingUtilitySelection = 4) AND NOT #StartBrine) OR ((#CoolingUtilitySelection = 5) AND #StartChilling AND NOT #StartBrine));
   #ChilledWaterOutletValve1 := #ChilledWaterInletValve1 AND NOT #StartJVDelay;
   #ChilledWaterInletValve2 := #ChilledWaterInletValve1 AND (#BatchSizeSel = 1);
   #ChilledWaterOutletValve2 := #ChilledWaterInletValve2 AND NOT #StartJVDelay;
   #BrineWaterInletValve1 := #_w7 AND ((#CoolingUtilitySelection = 2) OR ((#CoolingUtilitySelection = 4) AND #StartBrine) OR ((#CoolingUtilitySelection = 5) AND #StartBrine));
   #BrineWaterOutletValve1 := #BrineWaterInletValve1 AND NOT #StartJVDelay;
   #BrineWaterInletValve2 := #BrineWaterInletValve1 AND (#BatchSizeSel = 1);
   #BrineWaterOutletValve2 := #BrineWaterInletValve2 AND NOT #StartJVDelay;
   #BypassValve := #_w2 AND ((#StartUtility AND (#HeatTempReached OR #CoolTempReached)) OR NOT #StartUtility) AND #BypassSel;
   #JacketAirValve := #_w2 AND #StartJacketAirPurging;
   #_w8 := #_w1 AND #JacketPressureSelection AND NOT #JacketPressureReached AND NOT #JacketpressureTimer.TimeOver AND NOT #Temp;
   #JacketUtilityPressureValve := #_w8 AND (#JAcketActPressure < #JacketSafetyPressure);
   IF #_w8 AND (#JAcketActPressure >= #JacketSafetyPressure) THEN
       #JacketPressureReached := TRUE;
       #Temp := TRUE;
   END_IF;
END_REGION

REGION Network 16: Jacket Air Purging
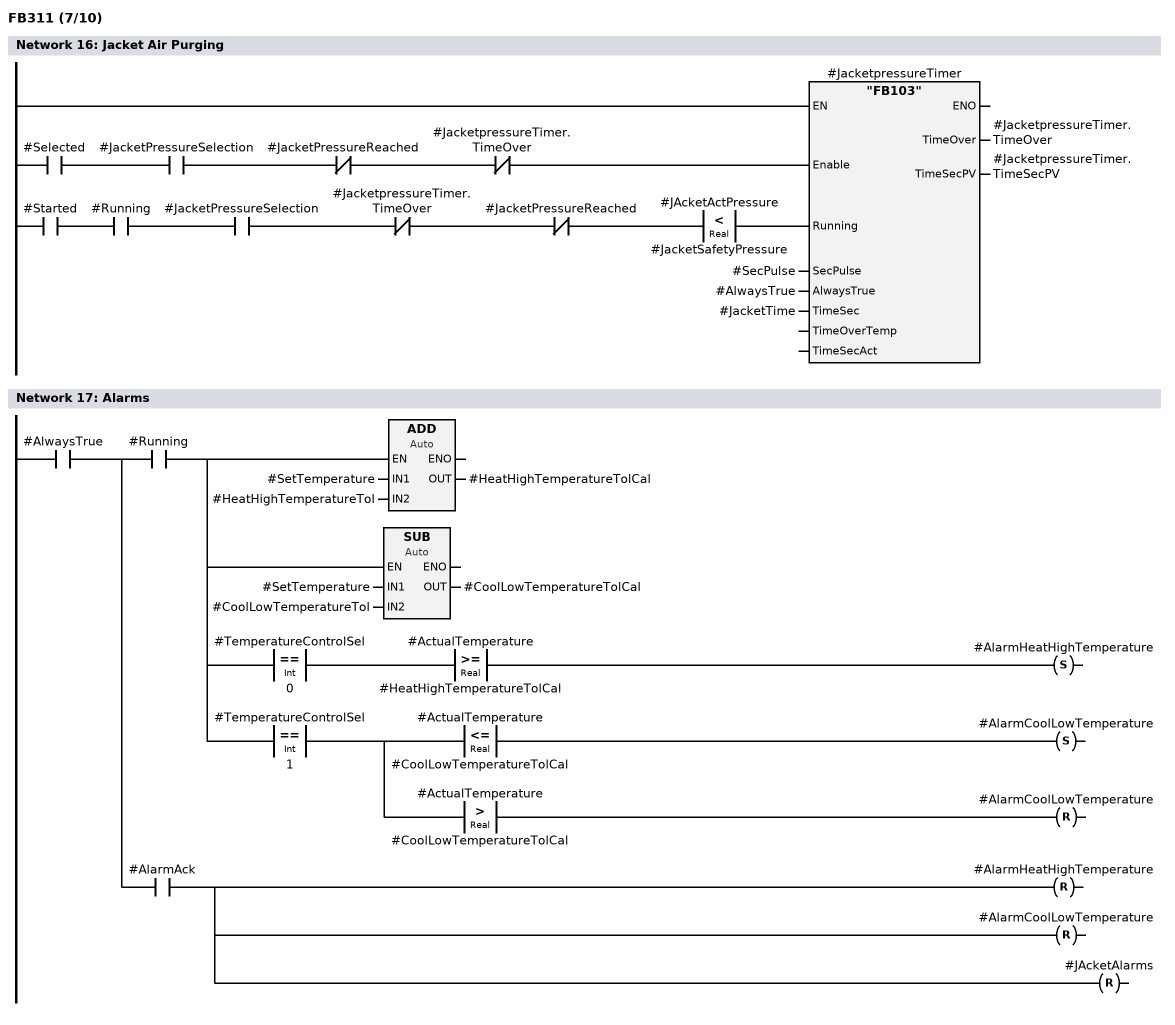
   RUNG wire#powerrail
      #JacketpressureTimer(Enable := wire#w1, Running := wire#w2, SecPulse := #SecPulse, AlwaysTrue := #AlwaysTrue, TimeSec := #JacketTime, TimeOverTemp :=, TimeSecAct :=, TimeOver => #JacketpressureTimer.TimeOver, TimeSecPV => #JacketpressureTimer.TimeSecPV)
   END_RUNG
   RUNG wire#powerrail
      Contact( #Selected )
      Contact( #JacketPressureSelection )
      I_Contact( #JacketPressureReached )
      I_Contact( #JacketpressureTimer.TimeOver )
   END_RUNG wire#w1
   RUNG wire#powerrail
      Contact( #Started )
      Contact( #Running )
      Contact( #JacketPressureSelection )
      I_Contact( #JacketpressureTimer.TimeOver )
      I_Contact( #JacketPressureReached )
      { S7_Templates := "SrcType := Real" } LT_Contact(in1 := #JAcketActPressure, in2 := #JacketSafetyPressure)
   END_RUNG wire#w2
   // the same network as SCL:
   #JacketpressureTimer(Enable := #Selected AND #JacketPressureSelection AND NOT #JacketPressureReached AND NOT #JacketpressureTimer.TimeOver,   // "FB103"
                        Running := #Started AND #Running AND #JacketPressureSelection AND NOT #JacketpressureTimer.TimeOver AND NOT #JacketPressureReached AND (#JAcketActPressure < #JacketSafetyPressure),
                        SecPulse := #SecPulse,
                        AlwaysTrue := #AlwaysTrue,
                        TimeSec := #JacketTime,
                        TimeOver => #JacketpressureTimer.TimeOver,
                        TimeSecPV => #JacketpressureTimer.TimeSecPV);
END_REGION

REGION Network 17: Alarms
   RUNG wire#powerrail
      Contact( #AlwaysTrue )
      wire#w1
      Contact( #Running )
      wire#w2
      Add(in1 := #SetTemperature, in2 := #HeatHighTemperatureTol, out => #HeatHighTemperatureTolCal)
   END_RUNG
   RUNG wire#w2
      Sub(in1 := #SetTemperature, in2 := #CoolLowTemperatureTol, out => #CoolLowTemperatureTolCal)
   END_RUNG
   RUNG wire#w2
      { S7_Templates := "SrcType := Int" } EQ_Contact(in1 := #TemperatureControlSel, in2 := 0)
      { S7_Templates := "SrcType := Real" } GE_Contact(in1 := #ActualTemperature, in2 := #HeatHighTemperatureTolCal)
      S_Coil( #AlarmHeatHighTemperature )
   END_RUNG
   RUNG wire#w2
      { S7_Templates := "SrcType := Int" } EQ_Contact(in1 := #TemperatureControlSel, in2 := 1)
      wire#w3
      { S7_Templates := "SrcType := Real" } LE_Contact(in1 := #ActualTemperature, in2 := #CoolLowTemperatureTolCal)
      S_Coil( #AlarmCoolLowTemperature )
   END_RUNG
   RUNG wire#w3
      { S7_Templates := "SrcType := Real" } GT_Contact(in1 := #ActualTemperature, in2 := #CoolLowTemperatureTolCal)
      R_Coil( #AlarmCoolLowTemperature )
   END_RUNG
   RUNG wire#w1
      Contact( #AlarmAck )
      wire#w4
      R_Coil( #AlarmHeatHighTemperature )
   END_RUNG
   RUNG wire#w4
      R_Coil( #AlarmCoolLowTemperature )
   END_RUNG
   RUNG wire#w4
      R_Coil( #JAcketAlarms )
   END_RUNG
   // the same network as SCL:
   #_w1 := #AlwaysTrue AND #Running;
   IF #_w1 THEN
       #HeatHighTemperatureTolCal := #SetTemperature + #HeatHighTemperatureTol;
       #CoolLowTemperatureTolCal := #SetTemperature - #CoolLowTemperatureTol;
   END_IF;
   IF #_w1 AND (#TemperatureControlSel = 0) AND (#ActualTemperature >= #HeatHighTemperatureTolCal) THEN
       #AlarmHeatHighTemperature := TRUE;
   END_IF;
   #_w2 := #_w1 AND (#TemperatureControlSel = 1);
   IF #_w2 AND (#ActualTemperature <= #CoolLowTemperatureTolCal) THEN
       #AlarmCoolLowTemperature := TRUE;
   END_IF;
   IF #_w2 AND (#ActualTemperature > #CoolLowTemperatureTolCal) THEN
       #AlarmCoolLowTemperature := FALSE;
   END_IF;
   IF #AlwaysTrue AND #AlarmAck THEN
       #AlarmHeatHighTemperature := FALSE;
       #AlarmCoolLowTemperature := FALSE;
       #JAcketAlarms := FALSE;
   END_IF;
END_REGION

REGION Network 18: Event Status
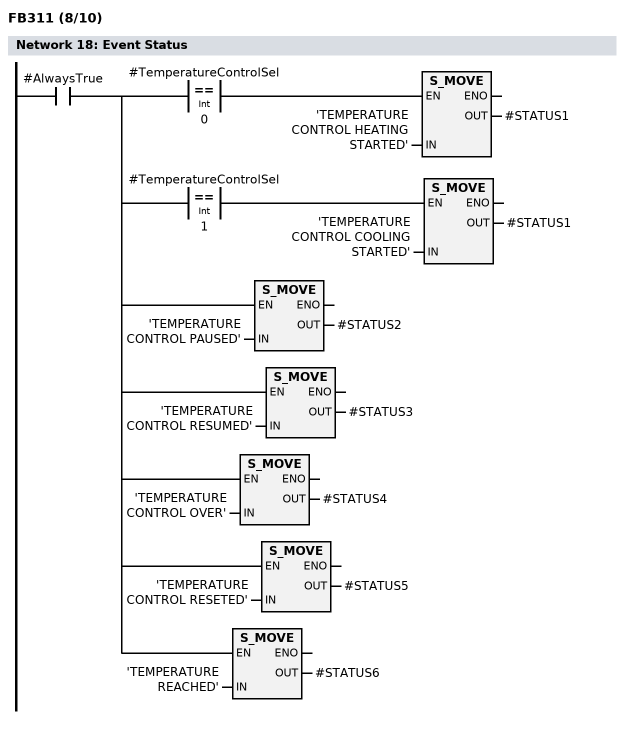
   RUNG wire#powerrail
      Contact( #AlwaysTrue )
      wire#w1
      { S7_Templates := "SrcType := Int" } EQ_Contact(in1 := #TemperatureControlSel, in2 := 0)
      S_Move(in := 'TEMPERATURE CONTROL HEATING STARTED', out => #STATUS1)
   END_RUNG
   RUNG wire#w1
      { S7_Templates := "SrcType := Int" } EQ_Contact(in1 := #TemperatureControlSel, in2 := 1)
      S_Move(in := 'TEMPERATURE CONTROL COOLING STARTED', out => #STATUS1)
   END_RUNG
   RUNG wire#w1
      S_Move(in := 'TEMPERATURE CONTROL PAUSED', out => #STATUS2)
   END_RUNG
   RUNG wire#w1
      S_Move(in := 'TEMPERATURE CONTROL RESUMED', out => #STATUS3)
   END_RUNG
   RUNG wire#w1
      S_Move(in := 'TEMPERATURE CONTROL OVER', out => #STATUS4)
   END_RUNG
   RUNG wire#w1
      S_Move(in := 'TEMPERATURE CONTROL RESETED', out => #STATUS5)
   END_RUNG
   RUNG wire#w1
      S_Move(in := 'TEMPERATURE REACHED', out => #STATUS6)
   END_RUNG
   // the same network as SCL:
   IF #AlwaysTrue AND (#TemperatureControlSel = 0) THEN
       #STATUS1 := 'TEMPERATURE CONTROL HEATING STARTED';
   END_IF;
   IF #AlwaysTrue AND (#TemperatureControlSel = 1) THEN
       #STATUS1 := 'TEMPERATURE CONTROL COOLING STARTED';
   END_IF;
   IF #AlwaysTrue THEN
       #STATUS2 := 'TEMPERATURE CONTROL PAUSED';
       #STATUS3 := 'TEMPERATURE CONTROL RESUMED';
       #STATUS4 := 'TEMPERATURE CONTROL OVER';
       #STATUS5 := 'TEMPERATURE CONTROL RESETED';
       #STATUS6 := 'TEMPERATURE REACHED';
   END_IF;
END_REGION

REGION Network 19: Print Logic
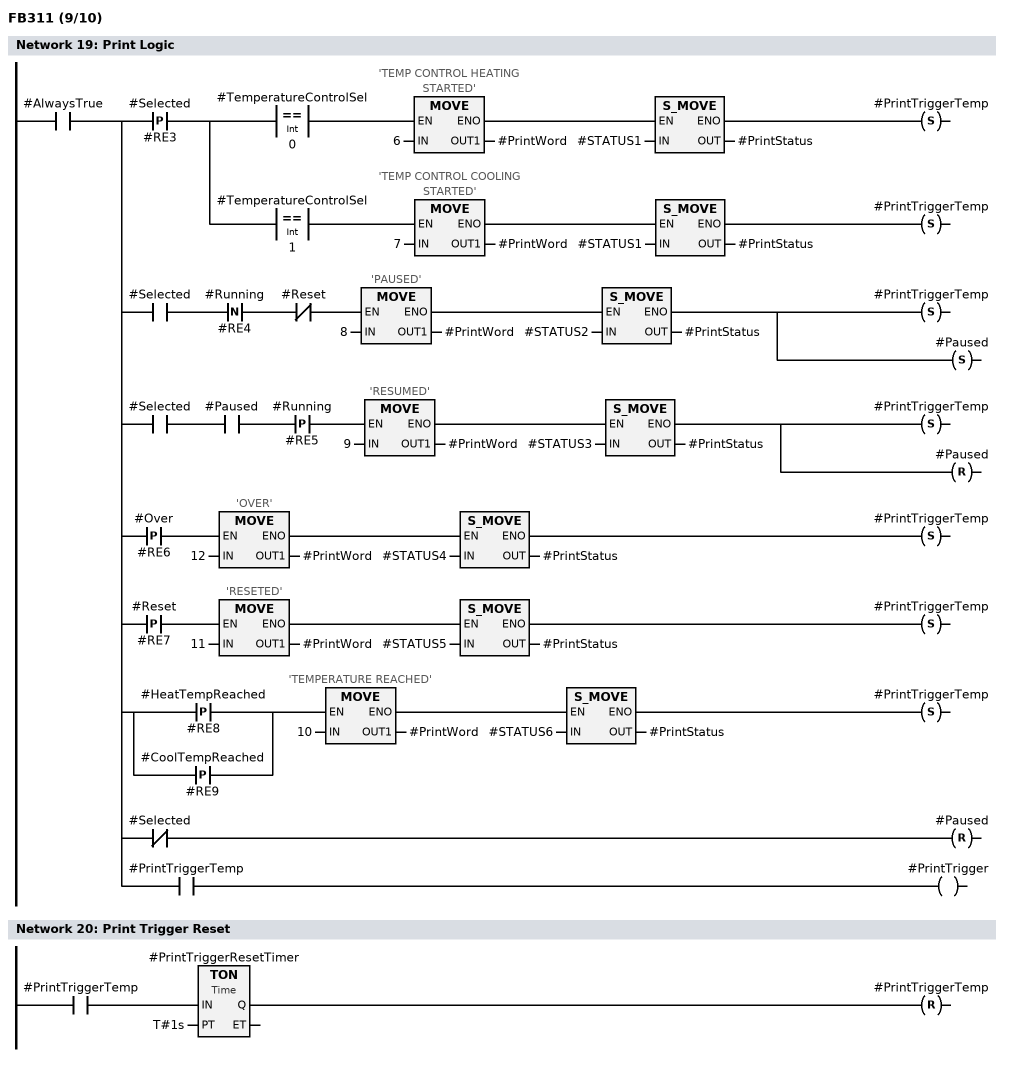
   RUNG wire#powerrail
      Contact( #AlwaysTrue )
      wire#w1
      P_Contact(operand := #Selected, bit := #RE3)
      wire#w2
      { S7_Templates := "SrcType := Int" } EQ_Contact(in1 := #TemperatureControlSel, in2 := 0)
      { S7_GenerateENO := "TRUE" } Move(in := 6, out1 => #PrintWord)   // 'TEMP CONTROL HEATING STARTED'
      S_Move(in := #STATUS1, out => #PrintStatus)
      S_Coil( #PrintTriggerTemp )
   END_RUNG
   RUNG wire#w2
      { S7_Templates := "SrcType := Int" } EQ_Contact(in1 := #TemperatureControlSel, in2 := 1)
      { S7_GenerateENO := "TRUE" } Move(in := 7, out1 => #PrintWord)   // 'TEMP CONTROL COOLING STARTED'
      S_Move(in := #STATUS1, out => #PrintStatus)
      S_Coil( #PrintTriggerTemp )
   END_RUNG
   RUNG wire#w1
      Contact( #Selected )
      N_Contact(operand := #Running, bit := #RE4)
      I_Contact( #Reset )
      { S7_GenerateENO := "TRUE" } Move(in := 8, out1 => #PrintWord)   // 'PAUSED'
      S_Move(in := #STATUS2, out => #PrintStatus)
      wire#w3
      S_Coil( #PrintTriggerTemp )
   END_RUNG
   RUNG wire#w3
      S_Coil( #Paused )
   END_RUNG
   RUNG wire#w1
      Contact( #Selected )
      Contact( #Paused )
      P_Contact(operand := #Running, bit := #RE5)
      { S7_GenerateENO := "TRUE" } Move(in := 9, out1 => #PrintWord)   // 'RESUMED'
      S_Move(in := #STATUS3, out => #PrintStatus)
      wire#w4
      S_Coil( #PrintTriggerTemp )
   END_RUNG
   RUNG wire#w4
      R_Coil( #Paused )
   END_RUNG
   RUNG wire#w1
      P_Contact(operand := #Over, bit := #RE6)
      { S7_GenerateENO := "TRUE" } Move(in := 12, out1 => #PrintWord)   // 'OVER'
      S_Move(in := #STATUS4, out => #PrintStatus)
      S_Coil( #PrintTriggerTemp )
   END_RUNG
   RUNG wire#w1
      P_Contact(operand := #Reset, bit := #RE7)
      { S7_GenerateENO := "TRUE" } Move(in := 11, out1 => #PrintWord)   // 'RESETED'
      S_Move(in := #STATUS5, out => #PrintStatus)
      S_Coil( #PrintTriggerTemp )
   END_RUNG
   RUNG wire#w1
      P_Contact(operand := #HeatTempReached, bit := #RE8)
      wire#w5
      { S7_GenerateENO := "TRUE" } Move(in := 10, out1 => #PrintWord)   // 'TEMPERATURE REACHED'
      S_Move(in := #STATUS6, out => #PrintStatus)
      S_Coil( #PrintTriggerTemp )
   END_RUNG
   RUNG wire#w1
      P_Contact(operand := #CoolTempReached, bit := #RE9)
   END_RUNG wire#w5
   RUNG wire#w1
      I_Contact( #Selected )
      R_Coil( #Paused )
   END_RUNG
   RUNG wire#w1
      Contact( #PrintTriggerTemp )
      Coil( #PrintTrigger )
   END_RUNG
   // the same network as SCL:
   // ENO of a box is taken as its EN; it also drops when the box reports an error
   #_w1 := #AlwaysTrue AND #Selected AND NOT #RE3;   // rising edge of #Selected
   #RE3 := #Selected;
   IF #_w1 AND (#TemperatureControlSel = 0) THEN
       #PrintWord := 6;   // 'TEMP CONTROL HEATING STARTED'
       #PrintStatus := #STATUS1;
       #PrintTriggerTemp := TRUE;
   END_IF;
   IF #_w1 AND (#TemperatureControlSel = 1) THEN
       #PrintWord := 7;   // 'TEMP CONTROL COOLING STARTED'
       #PrintStatus := #STATUS1;
       #PrintTriggerTemp := TRUE;
   END_IF;
   #_w2 := #AlwaysTrue AND #Selected AND NOT #Running AND #RE4;   // falling edge of #Running
   #RE4 := #Running;
   IF #_w2 AND NOT #Reset THEN
       #PrintWord := 8;   // 'PAUSED'
       #PrintStatus := #STATUS2;
       #PrintTriggerTemp := TRUE;
       #Paused := TRUE;
   END_IF;
   #_w3 := #AlwaysTrue AND #Selected AND #Paused AND #Running AND NOT #RE5;   // rising edge of #Running
   #RE5 := #Running;
   IF #_w3 THEN
       #PrintWord := 9;   // 'RESUMED'
       #PrintStatus := #STATUS3;
       #PrintTriggerTemp := TRUE;
       #Paused := FALSE;
   END_IF;
   #_w4 := #AlwaysTrue AND #Over AND NOT #RE6;   // rising edge of #Over
   #RE6 := #Over;
   IF #_w4 THEN
       #PrintWord := 12;   // 'OVER'
       #PrintStatus := #STATUS4;
       #PrintTriggerTemp := TRUE;
   END_IF;
   #_w5 := #AlwaysTrue AND #Reset AND NOT #RE7;   // rising edge of #Reset
   #RE7 := #Reset;
   IF #_w5 THEN
       #PrintWord := 11;   // 'RESETED'
       #PrintStatus := #STATUS5;
       #PrintTriggerTemp := TRUE;
   END_IF;
   #_w6 := #AlwaysTrue AND #HeatTempReached AND NOT #RE8;   // rising edge of #HeatTempReached
   #RE8 := #HeatTempReached;
   #_w7 := #AlwaysTrue AND #CoolTempReached AND NOT #RE9;   // rising edge of #CoolTempReached
   #RE9 := #CoolTempReached;
   IF #_w6 OR #_w7 THEN
       #PrintWord := 10;   // 'TEMPERATURE REACHED'
       #PrintStatus := #STATUS6;
       #PrintTriggerTemp := TRUE;
   END_IF;
   IF #AlwaysTrue AND NOT #Selected THEN #Paused := FALSE; END_IF;
   #PrintTrigger := #AlwaysTrue AND #PrintTriggerTemp;
END_REGION

REGION Network 20: Print Trigger Reset
   RUNG wire#powerrail
      Contact( #PrintTriggerTemp )
      { S7_Templates := "time_type := Time" } #PrintTriggerResetTimer.TON(pt := T#1s, et =>)
      R_Coil( #PrintTriggerTemp )
   END_RUNG
   // the same network as SCL:
   #PrintTriggerResetTimer(IN := #PrintTriggerTemp, PT := T#1s);   // TON
   IF #PrintTriggerResetTimer.Q THEN #PrintTriggerTemp := FALSE; END_IF;
END_REGION

REGION Network 21: Button Reset
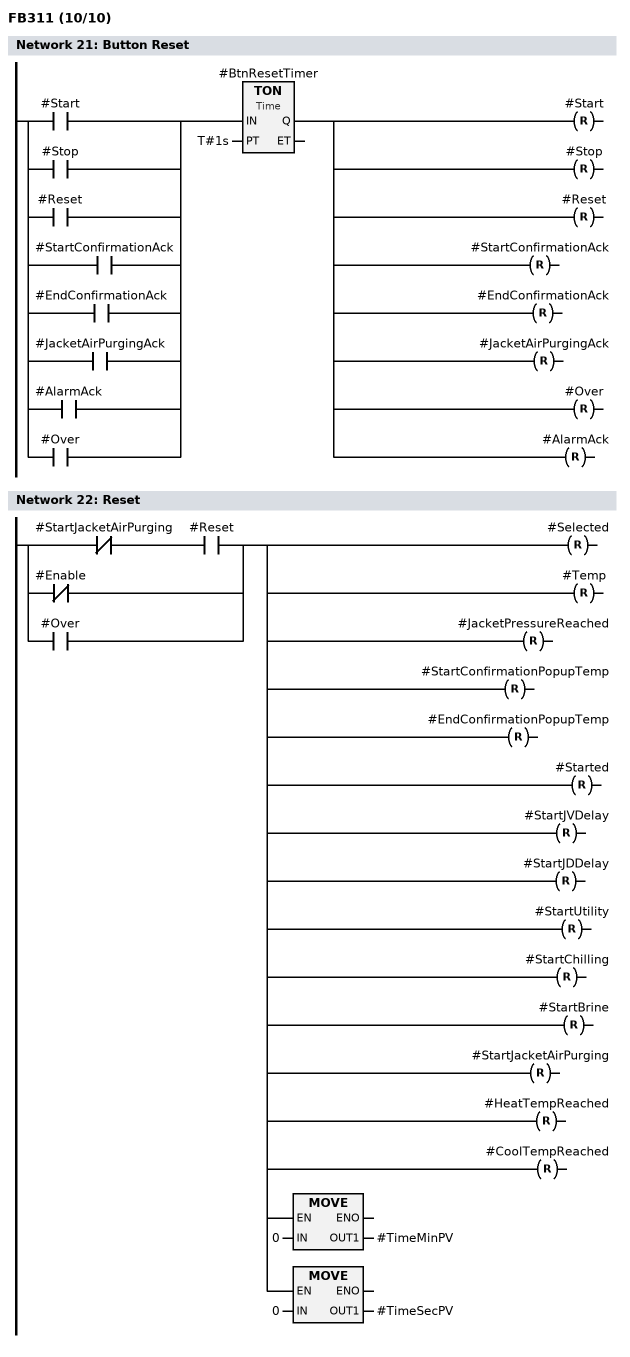
   RUNG wire#powerrail
      Contact( #Start )
      wire#w1
      { S7_Templates := "time_type := Time" } #BtnResetTimer.TON(pt := T#1s, et =>)
      wire#w2
      R_Coil( #Start )
   END_RUNG
   RUNG wire#powerrail
      Contact( #Stop )
   END_RUNG wire#w1
   RUNG wire#powerrail
      Contact( #Reset )
   END_RUNG wire#w1
   RUNG wire#powerrail
      Contact( #StartConfirmationAck )
   END_RUNG wire#w1
   RUNG wire#powerrail
      Contact( #EndConfirmationAck )
   END_RUNG wire#w1
   RUNG wire#powerrail
      Contact( #JacketAirPurgingAck )
   END_RUNG wire#w1
   RUNG wire#powerrail
      Contact( #AlarmAck )
   END_RUNG wire#w1
   RUNG wire#powerrail
      Contact( #Over )
   END_RUNG wire#w1
   RUNG wire#w2
      R_Coil( #Stop )
   END_RUNG
   RUNG wire#w2
      R_Coil( #Reset )
   END_RUNG
   RUNG wire#w2
      R_Coil( #StartConfirmationAck )
   END_RUNG
   RUNG wire#w2
      R_Coil( #EndConfirmationAck )
   END_RUNG
   RUNG wire#w2
      R_Coil( #JacketAirPurgingAck )
   END_RUNG
   RUNG wire#w2
      R_Coil( #Over )
   END_RUNG
   RUNG wire#w2
      R_Coil( #AlarmAck )
   END_RUNG
   // the same network as SCL:
   #BtnResetTimer(IN := #Start OR #Stop OR #Reset OR #StartConfirmationAck OR #EndConfirmationAck OR #JacketAirPurgingAck OR #AlarmAck OR #Over,   // TON
                  PT := T#1s);
   IF #BtnResetTimer.Q THEN
       #Start := FALSE;
       #Stop := FALSE;
       #Reset := FALSE;
       #StartConfirmationAck := FALSE;
       #EndConfirmationAck := FALSE;
       #JacketAirPurgingAck := FALSE;
       #Over := FALSE;
       #AlarmAck := FALSE;
   END_IF;
END_REGION

REGION Network 22: Reset
   RUNG wire#powerrail
      I_Contact( #StartJacketAirPurging )
      Contact( #Reset )
      wire#w1
      R_Coil( #Selected )
   END_RUNG
   RUNG wire#powerrail
      I_Contact( #Enable )
   END_RUNG wire#w1
   RUNG wire#powerrail
      Contact( #Over )
   END_RUNG wire#w1
   RUNG wire#w1
      R_Coil( #Temp )
   END_RUNG
   RUNG wire#w1
      R_Coil( #JacketPressureReached )
   END_RUNG
   RUNG wire#w1
      R_Coil( #StartConfirmationPopupTemp )
   END_RUNG
   RUNG wire#w1
      R_Coil( #EndConfirmationPopupTemp )
   END_RUNG
   RUNG wire#w1
      R_Coil( #Started )
   END_RUNG
   RUNG wire#w1
      R_Coil( #StartJVDelay )
   END_RUNG
   RUNG wire#w1
      R_Coil( #StartJDDelay )
   END_RUNG
   RUNG wire#w1
      R_Coil( #StartUtility )
   END_RUNG
   RUNG wire#w1
      R_Coil( #StartChilling )
   END_RUNG
   RUNG wire#w1
      R_Coil( #StartBrine )
   END_RUNG
   RUNG wire#w1
      R_Coil( #StartJacketAirPurging )
   END_RUNG
   RUNG wire#w1
      R_Coil( #HeatTempReached )
   END_RUNG
   RUNG wire#w1
      R_Coil( #CoolTempReached )
   END_RUNG
   RUNG wire#w1
      { S7_GenerateENO := "TRUE" } Move(in := 0, out1 => #TimeMinPV)
   END_RUNG
   RUNG wire#w1
      { S7_GenerateENO := "TRUE" } Move(in := 0, out1 => #TimeSecPV)
   END_RUNG
   // the same network as SCL:
   IF (NOT #StartJacketAirPurging AND #Reset) OR NOT #Enable OR #Over THEN
       #Selected := FALSE;
       #Temp := FALSE;
       #JacketPressureReached := FALSE;
       #StartConfirmationPopupTemp := FALSE;
       #EndConfirmationPopupTemp := FALSE;
       #Started := FALSE;
       #StartJVDelay := FALSE;
       #StartJDDelay := FALSE;
       #StartUtility := FALSE;
       #StartChilling := FALSE;
       #StartBrine := FALSE;
   END_IF;
   #_w1 := (NOT #StartJacketAirPurging AND #Reset) OR NOT #Enable OR #Over;
   IF #_w1 THEN
       #StartJacketAirPurging := FALSE;
       #HeatTempReached := FALSE;
       #CoolTempReached := FALSE;
       #TimeMinPV := 0;
       #TimeSecPV := 0;
   END_IF;
END_REGION
END_FUNCTION_BLOCK
